FUNCTION_BLOCK FB_Vise_Station
VAR_INPUT
	sName						:STRING;
	bEn							:BOOL;
	bEHA						:BOOL;
	bManualMode					:BOOL;
	bAck						:BOOL;
	sSourceName					:STRING(10);
	stViseBasePosEvent			:TcEventEntry;		(*Event definition*)
	stViseWorkPosEvent			:TcEventEntry;		(*Event definition*)
	stStopperInWorkPosEvent		:TcEventEntry;		(*Event definition*)
	stStopperOutWorkPosEvent	:TcEventEntry;		(*Event definition*)
	stViseStationSensors		:ST_Vise_Sensors;
END_VAR
VAR_OUTPUT
	bError 						:BOOL;
END_VAR
VAR
	fbVise						:FB_Bistabil;
	fbStopper_In				:FB_Bistabil;
	fbStopper_Out				:FB_Bistabil;
END_VAR

fbVise(
	sName:= sName,
	bEn:= bEn,						// AND fbStopper_In.bWorkPosStab,				Miért ?????????????????????????????????????????
	bEHA:= bEHA, 
	bDisableManualCmd:= NOT (bManualMode AND fbStopper_In.bWorkPosStab), 
	bAck:= bAckP,
	sSourceName:= sSourceName, 
	i_bBasePos:= stViseStationSensors.bViseIn,
	i_bWorkPos:= stViseStationSensors.bViseOut,
	stBasePosEvent:= stViseBasePosEvent,
	stWorkPosEvent:= stViseWorkPosEvent);
	
fbStopper_In(
	sName:= sName, 
	bEn:= bEn, 
	bEHA:= bEHA, 
	bDisableManualCmd:= NOT bManualMode, 
	bAck:= bAckP, 
	sSourceName:= sSourceName,
	i_bBasePos:= stViseStationSensors.bStopper_In_Release,
	i_bWorkPos:= stViseStationSensors.bStopper_In_Hold,
	stBasePosEvent:= TC_Events.MyEvents.Event,
	stWorkPosEvent:= stStopperInWorkPosEvent);

fbStopper_Out(
	sName:= sName, 
	bEn:= bEn, 
	bEHA:= bEHA, 
	bDisableManualCmd:= NOT bManualMode, 
	bAck:= bAckP, 
	sSourceName:= sSourceName,
	i_bBasePos:= stViseStationSensors.bStopper_Out_Release,
	i_bWorkPos:= stViseStationSensors.bStopper_Out_Hold,
	stBasePosEvent:= TC_Events.MyEvents.Event,
	stWorkPosEvent:= stStopperOutWorkPosEvent);
	
bError := fbStopper_In.bError OR fbStopper_Out.bError OR fbVise.bError;

PROPERTY PUBLIC StopperInner : REFERENCE TO FB_Bistabil
GET
StopperInner REF= fbStopper_In;
END_GET
END_PROPERTY

PROPERTY PUBLIC StopperOuter : REFERENCE TO FB_Bistabil
GET
StopperOuter REF= fbStopper_Out;
END_GET
END_PROPERTY

PROPERTY PUBLIC Vise : REFERENCE TO FB_Bistabil
GET
Vise REF= fbVise;
END_GET
END_PROPERTY

END_FUNCTION_BLOCK

(* stored: Version 1.1.0.1, ProductVersion 3.1.4024.11
   POU FB_Vise_Station: Id {dca77ff4-31c6-463b-b418-27516e63514d}, SpecialFunc None
   Property StopperInner: Id {7841bc5e-c2d5-4005-a558-b9137ecb09b9}
   Get Get: Id {a80d635b-7629-4407-836c-c734d04f00c0}
   Property StopperOuter: Id {c9d12e77-d4da-49f2-95f3-1f6cbdd86da3}
   Get Get: Id {607caa2b-f912-4499-be6d-cc7d834f1eda}
   Property Vise: Id {40939cac-d896-4760-a16b-644feb036ff8}
   Get Get: Id {c1a64b2a-e409-4af0-8e72-63c71b993edd} *)
